// TIA Portal V20 export
VAR_GLOBAL   // PLC tag table "Unit1Em2"
   "BA040AZSBK02.00" AT %I1004.0 : Bool;   // SUCTION PAD TOP UP
   "BA040AZSBK02.01" AT %I1004.1 : Bool;   // SUCTION PAD BTM DOWN
   "BA040AZSBK02.02" AT %I1004.2 : Bool;   // CUTTER DOWN
   "BA040AZSBK02.03" AT %I1004.3 : Bool;   // TAPE TOP UP
   "BA040AZSBK02.04" AT %I1004.4 : Bool;   // TAPE BTM DOWN
   "BA040AZSBK02.05" AT %I1004.5 : Bool;   // SPLICE HEAD ROTATE TOP BACKWARD
   "BA040AZSBK02.06" AT %I1004.6 : Bool;   // SPLICE HEAD ROTATE BTM BACKWARD
   "BA040AZSBK02.10" AT %I1005.0 : Bool;   // SUCTION PAD TOP DOWN
   "BA040AZSBK02.11" AT %I1005.1 : Bool;   // SUCTION PAD BTM UP
   "BA040AZSBK02.14" AT %I1005.4 : Bool;   // TAPE BTM UP
   "BA040AZSBK02.13" AT %I1005.3 : Bool;   // TAPE TOP DOWN
   "BA040AZSBK02.12" AT %I1005.2 : Bool;   // CUTTER UP
   "BA040AZSBK02.15" AT %I1005.5 : Bool;   // SPLICE HEAD ROTATE TOP FORWARD
   "BA040AZSBK02.16" AT %I1005.6 : Bool;   // SPLICE HEAD ROTATE BTM FORWARD
   "BA040AZSBK03.00" AT %I1008.0 : Bool;   // SUCTION PAD TOP LEFT PRESSURE SWITCH
   "BA040AZSBK03.01" AT %I1008.1 : Bool;   // SUCTION PAD TOP RIGHT PRESSURE SWITCH
   "BA040AZSBK03.02" AT %I1008.2 : Bool;   // SUCTION PAD BTM LEFT PRESSURE SWITCH
   "BA040AZSBK03.03" AT %I1008.3 : Bool;   // SUCTION PAD BTM RIGHT PRESSURE SWITCH
   "BA040AZSBK03.04" AT %I1008.4 : Bool;   // SUCTION PAD TOP TAPE PRESSURE SWITCH
   "BA040AZSBK03.05" AT %I1008.5 : Bool;   // SUCTION PAD BTM TAPE PRESSURE SWITCH
   "BA040AZSPM02.00" AT %Q2004.0 : Bool;   // SUCTION PAD #1 TOP DOWN
   "BA040AZSPM02.01" AT %Q2004.1 : Bool;   // SUCTION PAD #1 TOP UP
   "BA040AZSPM02.02" AT %Q2004.2 : Bool;   // SUCTION PAD #1 BTM UP
   "BA040AZSPM02.03" AT %Q2004.3 : Bool;   // SUCTION PAD #1 BTM DOWN
   "BA040AZSPM02.04" AT %Q2004.4 : Bool;   // CUTTER #1 UP
   "BA040AZSPM02.05" AT %Q2004.5 : Bool;   // CUTTER #1 DOWN
   "BA040AZSPM02.06" AT %Q2004.6 : Bool;   // TAPE #1 TOP DOWN
   "BA040AZSPM02.07" AT %Q2004.7 : Bool;   // TAPE #1 TOP UP
   "BA040AZSPM02.10" AT %Q2005.0 : Bool;   // TAPE #1 BTM UP
   "BA040AZSPM02.11" AT %Q2005.1 : Bool;   // TAPE #1 BTM DOWN
   "BA040AZSPM02.12" AT %Q2005.2 : Bool;   // SPLICE HEAD ROTATE #1 TOP FORWARD
   "BA040AZSPM02.13" AT %Q2005.3 : Bool;   // SPLICE HEAD ROTATE #1 TOP BACKWARD
   "BA040AZSPM02.14" AT %Q2005.4 : Bool;   // SPLICE HEAD ROTATE #1 BTM FORWARD
   "BA040AZSPM02.15" AT %Q2005.5 : Bool;   // SPLICE HEAD ROTATE #1 BTM BACKWARD
   "BA040AZSBK29.00" AT %Q2100.0 : Bool;   // SUCTION PAD TOP LEFT VACUUM ON
   "BA040AZSBK29.01" AT %Q2100.1 : Bool;   // SUCTION PAD TOP LEFT VACUUM OFF
   "BA040AZSBK29.02" AT %Q2100.2 : Bool;   // SUCTION PAD TOP RIGHT VACUUM ON
   "BA040AZSBK29.03" AT %Q2100.3 : Bool;   // SUCTION PAD TOP RIGHT VACUUM OFF
   "BA040AZSBK29.04" AT %Q2100.4 : Bool;   // SUCTION PAD BTM LEFT VACUUM ON
   "BA040AZSBK29.05" AT %Q2100.5 : Bool;   // SUCTION PAD BTM LEFT VACUUM OFF
   "BA040AZSBK29.06" AT %Q2100.6 : Bool;   // SUCTION PAD BTM RIGHT VACUUM ON
   "BA040AZSBK29.07" AT %Q2100.7 : Bool;   // SUCTION PAD BTM RIGHT VACUUM OFF
   "BA040AZSBK30.00" AT %Q2104.0 : Bool;   // SUCTION PAD TOP TAPE VACUUM ON
   "BA040AZSBK30.01" AT %Q2104.1 : Bool;   // SUCTION PAD TOP TAPE VACUUM OFF
   "BA040AZSBK30.02" AT %Q2104.2 : Bool;   // SUCTION PAD BTM TAPE VACUUM ON
   "BA040AZSBK30.03" AT %Q2104.3 : Bool;   // SUCTION PAD BTM TAPE VACUUM OFF
END_VAR
VAR_GLOBAL CONSTANT   // user constants
   U1EM2_JOB01 : DInt := 1;
   U1EM2_JOB02 : DInt := 2;
   U1EM2_JOB03 : DInt := 3;
   U1EM2_JOB04 : DInt := 4;
   U1EM2_JOB05 : DInt := 5;
   U1EM2_JOB06 : DInt := 6;
   U1EM2_JOB07 : DInt := 7;
   U1EM2_JOB08 : DInt := 8;
   U1EM2_JOB09 : DInt := 9;
   U1EM2_JOB10 : DInt := 10;
   U1EM2_JOB11 : DInt := 11;
   U1EM2_JOB12 : DInt := 12;
   U1EM2_JOB13 : DInt := 13;
   U1EM2_JOB14 : DInt := 14;
   U1EM2_JOB15 : DInt := 15;
   U1EM2_JOB16 : DInt := 16;
   U1EM2_JOB17 : DInt := 17;
   U1EM2_JOB18 : DInt := 18;
   U1EM2_JOB19 : DInt := 19;
   U1EM2_JOB20 : DInt := 20;
   U1EM2_JOB21 : DInt := 21;
   U1EM2_JOB22 : DInt := 22;
   U1EM2_JOB23 : DInt := 23;
   U1EM2_JOB24 : DInt := 24;
   U1EM2_JOB25 : DInt := 25;
   U1EM2_JOB26 : DInt := 26;
   U1EM2_JOB27 : DInt := 27;
   U1EM2_JOB28 : DInt := 28;
   U1EM2_JOB29 : DInt := 29;
   U1EM2_JOB30 : DInt := 30;
   U1EM2_JOB31 : DInt := 31;
   U1EM2_JOB32 : DInt := 32;
   U1EM2_JOB33 : DInt := 33;
   U1EM2_JOB34 : DInt := 34;
   U1EM2_JOB35 : DInt := 35;
   U1EM2_JOB36 : DInt := 36;
   U1EM2_JOB37 : DInt := 37;
   U1EM2_JOB38 : DInt := 38;
   U1EM2_JOB39 : DInt := 39;
   U1EM2_JOB40 : DInt := 40;
   U1EM2_JOB41 : DInt := 41;
   U1EM2_JOB42 : DInt := 42;
   U1EM2_JOB43 : DInt := 43;
   U1EM2_JOB44 : DInt := 44;
   U1EM2_JOB45 : DInt := 45;
   U1EM2_JOB46 : DInt := 46;
   U1EM2_JOB47 : DInt := 47;
   U1EM2_JOB48 : DInt := 48;
   U1EM2_JOB49 : DInt := 49;
   U1EM2_JOB50 : DInt := 50;
   U1EM2_JOB51 : DInt := 51;
   U1EM2_JOB52 : DInt := 52;
   U1EM2_JOB53 : DInt := 53;
   U1EM2_JOB54 : DInt := 54;
   U1EM2_JOB55 : DInt := 55;
   U1EM2_JOB56 : DInt := 56;
   U1EM2_JOB57 : DInt := 57;
   U1EM2_JOB58 : DInt := 58;
   U1EM2_JOB59 : DInt := 59;
   U1EM2_JOB60 : DInt := 60;
   U1EM2_JOB61 : DInt := 61;
   U1EM2_JOB62 : DInt := 62;
   U1EM2_JOB63 : DInt := 63;
   U1EM2_JOB64 : DInt := 64;
   U1EM2_JOB65 : DInt := 65;
   U1EM2_JOB66 : DInt := 66;
   U1EM2_JOB67 : DInt := 67;
   U1EM2_JOB68 : DInt := 68;
   U1EM2_JOB69 : DInt := 69;
   U1EM2_JOB70 : DInt := 70;
   U1EM2_JOB71 : DInt := 71;
   U1EM2_JOB72 : DInt := 72;
   U1EM2_JOB73 : DInt := 73;
   U1EM2_JOB74 : DInt := 74;
   U1EM2_JOB75 : DInt := 75;
   U1EM2_JOB76 : DInt := 76;
   U1EM2_JOB77 : DInt := 77;
   U1EM2_JOB78 : DInt := 78;
   U1EM2_JOB79 : DInt := 79;
   U1EM2_JOB80 : DInt := 80;
   U1EM2_JOB81 : DInt := 81;
   U1EM2_JOB82 : DInt := 82;
   U1EM2_JOB83 : DInt := 83;
   U1EM2_JOB84 : DInt := 84;
   U1EM2_JOB85 : DInt := 85;
   U1EM2_JOB86 : DInt := 86;
   U1EM2_JOB87 : DInt := 87;
   U1EM2_JOB88 : DInt := 88;
   U1EM2_JOB89 : DInt := 89;
   U1EM2_JOB90 : DInt := 90;
   U1EM2_JOB91 : DInt := 91;
   U1EM2_JOB92 : DInt := 92;
   U1EM2_JOB93 : DInt := 93;
   U1EM2_JOB94 : DInt := 94;
   U1EM2_JOB95 : DInt := 95;
   U1EM2_JOB96 : DInt := 96;
   U1EM2_JOB97 : DInt := 97;
   U1EM2_JOB98 : DInt := 98;
   U1EM2_JOB99 : DInt := 99;
   U1EM2_SEQUENCE01 : Int := 1;
   U1EM2_SEQUENCE02 : Int := 2;
   U1EM2_SEQUENCE03 : Int := 3;
   U1EM2_SEQUENCE04 : Int := 4;
   U1EM2_SEQUENCE05 : Int := 5;
   U1EM2_SEQUENCE06 : Int := 6;
   U1EM2_SEQUENCE07 : Int := 7;
   U1EM2_SEQUENCE08 : Int := 8;
   U1EM2_SEQUENCE09 : Int := 9;
   U1EM2_SEQUENCE10 : Int := 10;
   U1EM2_SEQUENCE11 : Int := 11;
   U1EM2_SEQUENCE12 : Int := 12;
   U1EM2_SEQUENCE13 : Int := 13;
   U1EM2_SEQUENCE14 : Int := 14;
   U1EM2_SEQUENCE15 : Int := 15;
   U1EM2_SEQUENCE16 : Int := 16;
   U1EM2_SEQUENCE17 : Int := 17;
   U1EM2_SEQUENCE18 : Int := 18;
   U1EM2_SEQUENCE19 : Int := 19;
   U1EM2_SEQUENCE20 : Int := 20;
   U1EM2_SEQUENCE21 : Int := 21;
   U1EM2_SEQUENCE22 : Int := 22;
   U1EM2_SEQUENCE23 : Int := 23;
   U1EM2_SEQUENCE24 : Int := 24;
   U1EM2_SEQUENCE25 : Int := 25;
   U1EM2_SEQUENCE26 : Int := 26;
   U1EM2_SEQUENCE27 : Int := 27;
   U1EM2_SEQUENCE28 : Int := 28;
   U1EM2_SEQUENCE29 : Int := 29;
   U1EM2_SEQUENCE30 : Int := 30;
   U1EM2_SEQUENCE31 : Int := 31;
   U1EM2_SEQUENCE32 : Int := 32;
   U1EM2_SEQUENCE33 : Int := 33;
   U1EM2_SEQUENCE34 : Int := 34;
   U1EM2_SEQUENCE35 : Int := 35;
   U1EM2_SEQUENCE36 : Int := 36;
   U1EM2_SEQUENCE37 : Int := 37;
   U1EM2_SEQUENCE38 : Int := 38;
   U1EM2_SEQUENCE39 : Int := 39;
   U1EM2_SEQUENCE40 : Int := 40;
   U1EM2_SEQUENCE41 : Int := 41;
   U1EM2_SEQUENCE42 : Int := 42;
   U1EM2_SEQUENCE43 : Int := 43;
   U1EM2_SEQUENCE44 : Int := 44;
   U1EM2_SEQUENCE45 : Int := 45;
   U1EM2_SEQUENCE46 : Int := 46;
   U1EM2_SEQUENCE47 : Int := 47;
   U1EM2_SEQUENCE48 : Int := 48;
   U1EM2_SEQUENCE49 : Int := 49;
   U1EM2_SEQUENCE50 : Int := 50;
   U1EM2_SEQUENCE51 : Int := 51;
   U1EM2_SEQUENCE52 : Int := 52;
   U1EM2_SEQUENCE53 : Int := 53;
   U1EM2_SEQUENCE54 : Int := 54;
   U1EM2_SEQUENCE55 : Int := 55;
   U1EM2_SEQUENCE56 : Int := 56;
   U1EM2_SEQUENCE57 : Int := 57;
   U1EM2_SEQUENCE58 : Int := 58;
   U1EM2_SEQUENCE59 : Int := 59;
   U1EM2_SEQUENCE60 : Int := 60;
   U1EM2_SEQUENCE61 : Int := 61;
   U1EM2_SEQUENCE62 : Int := 62;
   U1EM2_SEQUENCE63 : Int := 63;
   U1EM2_SEQUENCE64 : Int := 64;
   U1EM2_SEQUENCE65 : Int := 65;
   U1EM2_SEQUENCE66 : Int := 66;
   U1EM2_SEQUENCE67 : Int := 67;
   U1EM2_SEQUENCE68 : Int := 68;
   U1EM2_SEQUENCE69 : Int := 69;
   U1EM2_SEQUENCE70 : Int := 70;
   U1EM2_SEQUENCE71 : Int := 71;
   U1EM2_SEQUENCE72 : Int := 72;
   U1EM2_SEQUENCE73 : Int := 73;
   U1EM2_SEQUENCE74 : Int := 74;
   U1EM2_SEQUENCE75 : Int := 75;
   U1EM2_SEQUENCE76 : Int := 76;
   U1EM2_SEQUENCE77 : Int := 77;
   U1EM2_SEQUENCE78 : Int := 78;
   U1EM2_SEQUENCE79 : Int := 79;
   U1EM2_SEQUENCE80 : Int := 80;
   U1EM2_SEQUENCE81 : Int := 81;
   U1EM2_SEQUENCE82 : Int := 82;
   U1EM2_SEQUENCE83 : Int := 83;
   U1EM2_SEQUENCE84 : Int := 84;
   U1EM2_SEQUENCE85 : Int := 85;
   U1EM2_SEQUENCE86 : Int := 86;
   U1EM2_SEQUENCE87 : Int := 87;
   U1EM2_SEQUENCE88 : Int := 88;
   U1EM2_SEQUENCE89 : Int := 89;
   U1EM2_SEQUENCE90 : Int := 90;
   U1EM2_SEQUENCE91 : Int := 91;
   U1EM2_SEQUENCE92 : Int := 92;
   U1EM2_SEQUENCE93 : Int := 93;
   U1EM2_SEQUENCE94 : Int := 94;
   U1EM2_SEQUENCE95 : Int := 95;
   U1EM2_SEQUENCE96 : Int := 96;
   U1EM2_SEQUENCE97 : Int := 97;
   U1EM2_SEQUENCE98 : Int := 98;
   U1EM2_SEQUENCE99 : Int := 99;
   U1EM2_NO_OF_SEQUENCE : USInt := 3;
END_VAR
